// TIA Portal V20 export
// export: Created 2025-12-01T14:56:17.3662073Z, ExportSetting None, DisplayName Totally Integrated Automation Portal, DisplayVersion V20 Update 3, DisplayName TIA Portal Openness, DisplayVersion V20 Update 3, DisplayName TIA Portal Version Control Interface, DisplayVersion V20 Update 3, DisplayName STEP 7 Professional, DisplayVersion V20 Update 3, DisplayName STEP 7 Safety, DisplayVersion V20 Update 2, DisplayName WinCC Basic/Comfort/Advanced, DisplayVersion V20 Update 3, DisplayName WinCC Professional, DisplayVersion V20 Update 3, DisplayName WinCC Unified, DisplayVersion V20 Update 3
TYPE "UDT_Interlock_manual_Puerta_Rapida"
   STRUCT
      "byte0.bit0" : Bool;
      "byte0.bit1" : Bool;
      "byte0.bit2" : Bool;
      "byte0.bit3" : Bool;
      "byte0.bit4" : Bool;
      "Byte0.bit5" : Bool;
      Abrir_Puerta : Bool;
      Cerrar_Puerta : Bool;
      Byte1_bit0 : Bool;
      Byte1_bit1 : Bool;
      Byte1_bit2 : Bool;
      Byte1_bit3 : Bool;
      Byte1_bit4 : Bool;
      Byte1_bit5 : Bool;
      Byte1_bit6 : Bool;
      Byte1_bit7 : Bool;
   END_STRUCT;
END_TYPE
